(* PLC project Generated.project, CODESYS CODESYS V3.5 SP19 Patch 1 *)
(* stored: creationDateTime 2026-09-01T00:57:57.899392, modificationDateTime 2026-09-01T00:57:57.899392 *)

(* ═══════════════════════════════════════════════════════════════ 🎮 ST_CycleDumpAtTremieCmd — Sélections IHM cycle vidage trémie (legacy) ═══════════════════════════════════════════════════════════════ *)
TYPE ST_CycleDumpAtTremieCmd : STRUCT
  TglEnableDumpAtTremie : BOOL := FALSE;  (* Mode vidage à la trémie — RESTREINT des mouvements dès le boot *)
END_STRUCT;
END_TYPE
